// TIA Portal project "2run-2stop-2motors" (V16)

(* hardware
DEVICE "S7-1200 station_1"  S7-1200 Station
   slot 0: "Rack_0"  S7-1200 Rack  Rack  V1.0
   slot 1: "PLC_1"  CPU 1212C AC/DC/Rly  6ES7 212-1BE40-0XB0  V4.0
*)

// ===== PLC "PLC_1"  CPU 1212C AC/DC/Rly =====

VAR_GLOBAL   // PLC tag table "Default tag table"
   "start" AT %I0.0 : Bool;
   "stop" AT %I0.1 : Bool;
   "km1" AT %Q0.0 : Bool;
   "km2" AT %Q0.1 : Bool;
   "loop marker" AT %M0.0 : Bool;
   "stage1break" AT %M0.1 : Bool;
   "stage2break" AT %M0.2 : Bool;
   "km2-ss" AT %M1.0 : Bool;
   "break1-ss" AT %M1.1 : Bool;
   "break2-ss" AT %M1.2 : Bool;
END_VAR

// folder: System blocks/Program resources

DATA_BLOCK "T1 5s"   // DB1
{ S7_Optimized_Access := 'TRUE' }
AUTHOR : Simatic
FAMILY : IEC
NAME : IEC_TMR
VERSION : 1.0
// stored: InstanceOfName IEC_TIMER
"IEC_TIMER"
BEGIN
END_DATA_BLOCK

DATA_BLOCK "T1 2s"   // DB2
{ S7_Optimized_Access := 'TRUE' }
AUTHOR : Simatic
FAMILY : IEC
NAME : IEC_TMR
VERSION : 1.0
// stored: InstanceOfName IEC_TIMER
"IEC_TIMER"
BEGIN
END_DATA_BLOCK

DATA_BLOCK "C1"   // DB3
{ S7_Optimized_Access := 'TRUE' }
AUTHOR : Simatic
FAMILY : IEC
NAME : CNTR
VERSION : 1.0
// stored: InstanceOfName IEC_COUNTER
"IEC_COUNTER"
BEGIN
END_DATA_BLOCK

DATA_BLOCK "T2 5s"   // DB4
{ S7_Optimized_Access := 'TRUE' }
AUTHOR : Simatic
FAMILY : IEC
NAME : IEC_TMR
VERSION : 1.0
// stored: InstanceOfName IEC_TIMER
"IEC_TIMER"
BEGIN
END_DATA_BLOCK

DATA_BLOCK "T2 2s"   // DB5
{ S7_Optimized_Access := 'TRUE' }
AUTHOR : Simatic
FAMILY : IEC
NAME : IEC_TMR
VERSION : 1.0
// stored: InstanceOfName IEC_TIMER
"IEC_TIMER"
BEGIN
END_DATA_BLOCK

DATA_BLOCK "C2"   // DB6
{ S7_Optimized_Access := 'TRUE' }
AUTHOR : Simatic
FAMILY : IEC
NAME : CNTR
VERSION : 1.0
// stored: InstanceOfName IEC_COUNTER
"IEC_COUNTER"
BEGIN
END_DATA_BLOCK

// folder: (top level)

ORGANIZATION_BLOCK "Main"   // OB1, LAD, ProgramCycle
TITLE = "Main Program Sweep (Cycle)"
{ S7_Optimized_Access := 'TRUE' }
VERSION : 0.1
   VAR_INPUT
      Initial_Call : Bool;   // Initial call of this OB
      Remanence : Bool;   // =True, if remanent data are available
   END_VAR
BEGIN

REGION Network 1
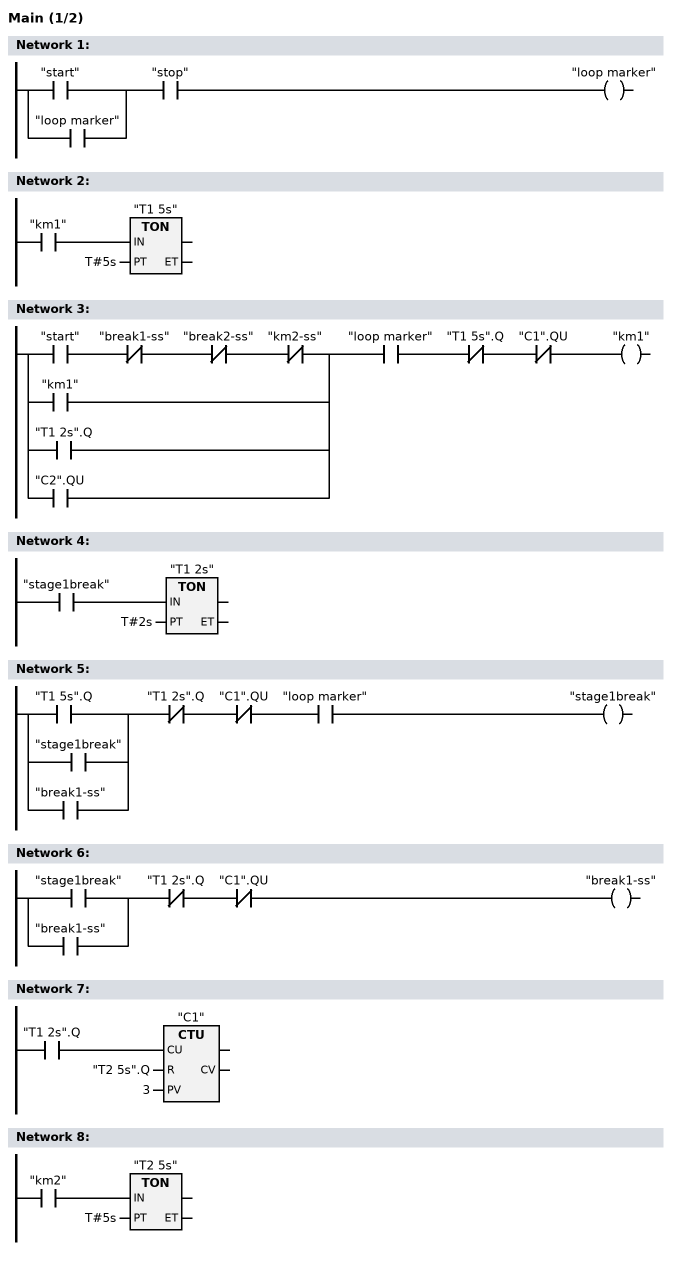
   RUNG wire#powerrail
      Contact( "start" )
      wire#w1
      Contact( "stop" )
      Coil( "loop marker" )
   END_RUNG
   RUNG wire#powerrail
      Contact( "loop marker" )
   END_RUNG wire#w1
   // the same network as SCL:
   "loop marker" := ("start" OR "loop marker") AND "stop";
END_REGION

REGION Network 2
   "T1 5s".TON(IN := "km1", PT := T#5s);
END_REGION

REGION Network 3
   RUNG wire#powerrail
      Contact( "start" )
      I_Contact( "break1-ss" )
      I_Contact( "break2-ss" )
      I_Contact( "km2-ss" )
      wire#w1
      Contact( "loop marker" )
      I_Contact( "T1 5s".Q )
      I_Contact( "C1".QU )
      Coil( "km1" )
   END_RUNG
   RUNG wire#powerrail
      Contact( "km1" )
   END_RUNG wire#w1
   RUNG wire#powerrail
      Contact( "T1 2s".Q )
   END_RUNG wire#w1
   RUNG wire#powerrail
      Contact( "C2".QU )
   END_RUNG wire#w1
   // the same network as SCL:
   "km1" := (("start" AND NOT "break1-ss" AND NOT "break2-ss" AND NOT "km2-ss") OR "km1" OR "T1 2s".Q OR "C2".QU) AND "loop marker" AND NOT "T1 5s".Q AND NOT "C1".QU;
END_REGION

REGION Network 4
   "T1 2s".TON(IN := "stage1break", PT := T#2s);
END_REGION

REGION Network 5
   RUNG wire#powerrail
      Contact( "T1 5s".Q )
      wire#w1
      I_Contact( "T1 2s".Q )
      I_Contact( "C1".QU )
      Contact( "loop marker" )
      Coil( "stage1break" )
   END_RUNG
   RUNG wire#powerrail
      Contact( "stage1break" )
   END_RUNG wire#w1
   RUNG wire#powerrail
      Contact( "break1-ss" )
   END_RUNG wire#w1
   // the same network as SCL:
   "stage1break" := ("T1 5s".Q OR "stage1break" OR "break1-ss") AND NOT "T1 2s".Q AND NOT "C1".QU AND "loop marker";
END_REGION

REGION Network 6
   RUNG wire#powerrail
      Contact( "stage1break" )
      wire#w1
      I_Contact( "T1 2s".Q )
      I_Contact( "C1".QU )
      Coil( "break1-ss" )
   END_RUNG
   RUNG wire#powerrail
      Contact( "break1-ss" )
   END_RUNG wire#w1
   // the same network as SCL:
   "break1-ss" := ("stage1break" OR "break1-ss") AND NOT "T1 2s".Q AND NOT "C1".QU;
END_REGION

REGION Network 7
   "C1".CTU(CU := "T1 2s".Q, R := "T2 5s".Q, PV := 3);
END_REGION

REGION Network 8
   "T2 5s".TON(IN := "km2", PT := T#5s);
END_REGION

REGION Network 9
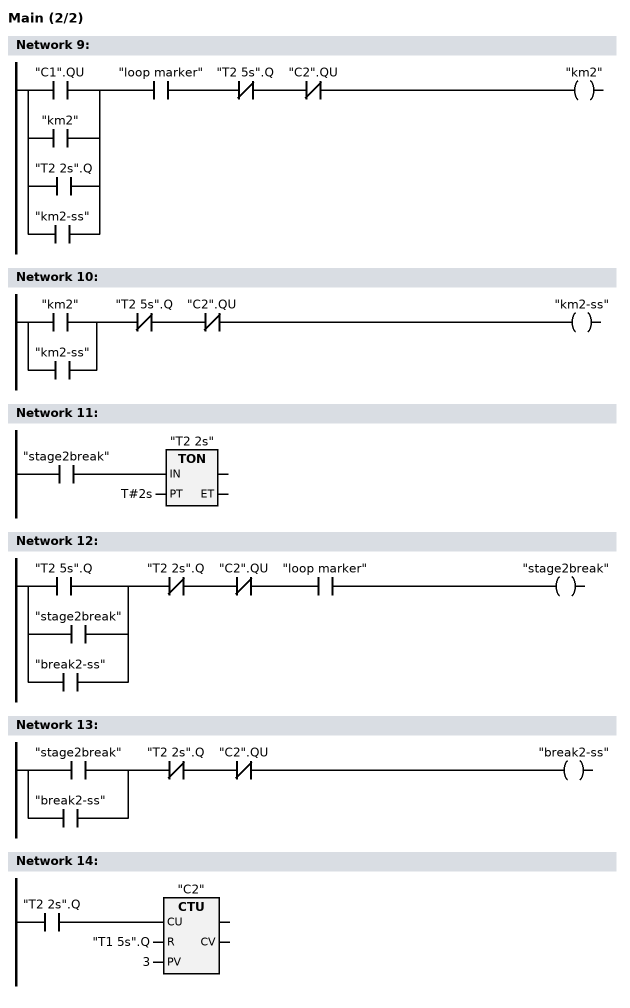
   RUNG wire#powerrail
      Contact( "C1".QU )
      wire#w1
      Contact( "loop marker" )
      I_Contact( "T2 5s".Q )
      I_Contact( "C2".QU )
      Coil( "km2" )
   END_RUNG
   RUNG wire#powerrail
      Contact( "km2" )
   END_RUNG wire#w1
   RUNG wire#powerrail
      Contact( "T2 2s".Q )
   END_RUNG wire#w1
   RUNG wire#powerrail
      Contact( "km2-ss" )
   END_RUNG wire#w1
   // the same network as SCL:
   "km2" := ("C1".QU OR "km2" OR "T2 2s".Q OR "km2-ss") AND "loop marker" AND NOT "T2 5s".Q AND NOT "C2".QU;
END_REGION

REGION Network 10
   RUNG wire#powerrail
      Contact( "km2" )
      wire#w1
      I_Contact( "T2 5s".Q )
      I_Contact( "C2".QU )
      Coil( "km2-ss" )
   END_RUNG
   RUNG wire#powerrail
      Contact( "km2-ss" )
   END_RUNG wire#w1
   // the same network as SCL:
   "km2-ss" := ("km2" OR "km2-ss") AND NOT "T2 5s".Q AND NOT "C2".QU;
END_REGION

REGION Network 11
   "T2 2s".TON(IN := "stage2break", PT := T#2s);
END_REGION

REGION Network 12
   RUNG wire#powerrail
      Contact( "T2 5s".Q )
      wire#w1
      I_Contact( "T2 2s".Q )
      I_Contact( "C2".QU )
      Contact( "loop marker" )
      Coil( "stage2break" )
   END_RUNG
   RUNG wire#powerrail
      Contact( "stage2break" )
   END_RUNG wire#w1
   RUNG wire#powerrail
      Contact( "break2-ss" )
   END_RUNG wire#w1
   // the same network as SCL:
   "stage2break" := ("T2 5s".Q OR "stage2break" OR "break2-ss") AND NOT "T2 2s".Q AND NOT "C2".QU AND "loop marker";
END_REGION

REGION Network 13
   RUNG wire#powerrail
      Contact( "stage2break" )
      wire#w1
      I_Contact( "T2 2s".Q )
      I_Contact( "C2".QU )
      Coil( "break2-ss" )
   END_RUNG
   RUNG wire#powerrail
      Contact( "break2-ss" )
   END_RUNG wire#w1
   // the same network as SCL:
   "break2-ss" := ("stage2break" OR "break2-ss") AND NOT "T2 2s".Q AND NOT "C2".QU;
END_REGION

REGION Network 14
   "C2".CTU(CU := "T2 2s".Q, R := "T1 5s".Q, PV := 3);
END_REGION
END_ORGANIZATION_BLOCK